(*
:Info: See <https://github.com/hganchev/twincat-tools/tree/main/TwinCAT%20Tools/twincat-tools/POUs/String/>
:Author: hganchev <https://github.com/hganchev/>

**Description:**

This function takes a string sInput and a split character sSplitChar and splits the input string into an array of substrings. 
The resulting array, F_STRING_SPLIT, has a size of Parameters.iSplitArraySize.

**Inputs:**

This function takes a string sInput and a split character sSplitChar and splits the input string into an array of substrings. 
The resulting array, F_STRING_SPLIT, has a size of Parameters.iSplitArraySize.

**Output:**

This implementation iteratively splits the input string using the specified split character. It assigns each substring to the corresponding element in the F_STRING_SPLIT array. 
The splitting process continues until either the end of the input string is reached or the maximum number of substrings specified by Parameters.iSplitArraySize is reached.

**Usage:**

.. code::

	VAR 
		sArray : ARRAY[0..Parameters.iSplitArraySize] OF STRING(255);
	END_VAR
	
	sArray := F_STRING_SPLIT(sInput := 'Hello,World', sSplitChar := ',');
	
Result:

sArray[0] = 'Hello'
sArray[1] = 'World'
*)

FUNCTION F_STRING_SPLIT : ARRAY[0..Parameters.iSplitArraySize] OF STRING(255)
VAR_INPUT
	sInput			: STRING(255);
	sSplitChar		: STRING(1);
END_VAR
VAR
	sCopy			: STRING(255);
	sSplit			: STRING(255);
	iDeleteLen		: INT;
	i				: INT;
END_VAR

sCopy := sInput;

FOR i := 0 TO Parameters.iSplitArraySize DO
	IF FIND(sCopy, sSplitChar) > 0 THEN
		sSplit := LEFT(sCopy, FIND(sCopy, sSplitChar) - 1);
		iDeleteLen := LEN(sSplit) + LEN(sSplitChar);
	ELSE
		sSplit := sCopy;
		iDeleteLen := LEN(sSplit);
	END_IF
	
	// Take the string value
	F_STRING_SPLIT[i] := sSplit;
	
	// Delete 
	sCopy := DELETE(sCopy, iDeleteLen, 1);
	
	// End of split
	IF sCopy = '' THEN
		EXIT;
	END_IF
END_FOR

END_FUNCTION

(* stored: Version 1.1.0.1, ProductVersion 3.1.4024.9
   POU F_STRING_SPLIT: Id {bf09d747-8a2c-4de8-9a8b-909da6c686c1}, SpecialFunc None *)
